FUNCTION_BLOCK MoveModuloMoverToPosition EXTENDS TaskBase
VAR_INPUT
END_VAR
VAR_OUTPUT
END_VAR
VAR
	moveAbs	: MC_MoveAbsoluteCA;
	_axis : REFERENCE TO AXIS_REF;
	_MoveMover : BOOL;
	_stOptions : ST_MoveAbsoluteCAOptions;
END_VAR

METHOD Abort : BOOL
moveAbs.Execute := FALSE;
moveAbs.Position := moveAbs.Velocity := 0;
_MoveMover := false;
_busy := false;
Abort := true;
State := 0;
END_METHOD

PROPERTY PUBLIC Acceleration : mc_lreal
GET
Acceleration := moveAbs.Acceleration;
END_GET
SET
moveAbs.Acceleration := Acceleration;
END_SET
END_PROPERTY

METHOD Cycle : BOOL
VAR_INPUT
END_VAR
CASE State OF
	0:
		IF _MoveMover THEN
			_done := FALSE;
			_error := FALSE;
			_busy := TRUE;
			moveAbs.Execute := TRUE;
			IF moveAbs.Busy THEN
				State := 10;
				_MoveMover := FALSE;
			END_IF
		END_IF
		
	10:
		IF NOT moveAbs.Busy THEN
			IF moveAbs.Done THEN
				_done := TRUE;
			ELSIF moveAbs.Error THEN
				_error := TRUE;
			END_IF
			_busy := FALSE;
			moveAbs.Execute := FALSE;
			State := 0;
		END_IF
END_CASE

moveAbs(Axis := _axis, Options := _stOptions);
END_METHOD

PROPERTY PUBLIC Deceleration : mc_lreal
GET
Deceleration := moveAbs.Deceleration;
END_GET
SET
moveAbs.Deceleration := Deceleration;
END_SET
END_PROPERTY

METHOD FB_init : BOOL
VAR_INPUT
	bInitRetains : BOOL; // if TRUE, the retain variables are initialized (warm start / cold start)
	bInCopyCode : BOOL;  // if TRUE, the instance afterwards gets moved into the copy code (online change)
	axis : reference TO AXIS_REF;
END_VAR
_axis REF= axis;
END_METHOD

PROPERTY PUBLIC Gap : mc_lreal
GET
Gap := moveAbs.Gap;
END_GET
SET
moveAbs.Gap := Gap;
END_SET
END_PROPERTY

PROPERTY PUBLIC Jerk : mc_lreal
GET
Jerk := moveAbs.Jerk;
END_GET
SET
moveAbs.Jerk := Jerk;
END_SET
END_PROPERTY

METHOD MoveTo : BOOL
VAR_INPUT
	Position : MC_LREAL;
	Velocity : MC_LREAL;
	Direction: Tc3_Mc3Definitions.MC_DIRECTION;
	Turns: UDINT;
END_VAR
moveAbs.Position := Position;
moveAbs.Velocity := Velocity;
moveAbs.Direction := Direction;
moveAbs.Options.AdditionalTurns := Turns;
_MoveMover := MoveTo := true;
END_METHOD

PROPERTY PUBLIC Options : ST_MoveAbsoluteCAOptions
GET
Options := _stOptions;
END_GET
SET
_stOptions := Options;
END_SET
END_PROPERTY

END_FUNCTION_BLOCK

(* stored: Version 1.1.0.1, ProductVersion 3.1.4024.12
   POU MoveModuloMoverToPosition: Id {996fe608-f005-43b0-b7bb-f33f237511c5}, SpecialFunc None
   Method Abort: Id {e91f53d6-3fee-47da-b969-b12290444a1f}
   Property Acceleration: Id {9cca71bc-09f7-4ec5-a9e0-372ce880866d}
   Get Get: Id {8efab319-7a15-4b02-96d3-afb30733e7b6}
   Set Set: Id {7f6e5164-788c-42d5-9777-9034d8aee40a}
   Method Cycle: Id {17422f94-11d5-4870-b9cb-2971dc153481}
   Property Deceleration: Id {844ebaf1-91dd-4442-8c33-92bcbeac6dea}
   Get Get: Id {50b8d5dc-c5e8-49f1-8033-680b16568e17}
   Set Set: Id {c1fd28c1-52e9-40a5-a51c-7d8bad271f43}
   Method FB_init: Id {37d409ee-dd67-4ea2-bddf-a65d46cc40e5}
   Property Gap: Id {1f9f5e65-07fb-4eac-aedb-feef80486e30}
   Get Get: Id {67ac09b0-11e2-4124-826d-72346d915abb}
   Set Set: Id {62c5bf39-3859-4737-8183-2c2206b5176d}
   Property Jerk: Id {cce85ebc-6201-45ef-a6f2-00296f696976}
   Get Get: Id {9dd7b014-e337-43e8-be50-6abb225db838}
   Set Set: Id {dcb14394-7c86-41b4-80fe-e9c7416faef5}
   Method MoveTo: Id {457265c4-5c25-4ff8-a5c9-719e58c0811a}
   Property Options: Id {c95271b4-8041-4fcf-9fb6-4915363c060f}
   Get Get: Id {965704cd-ef53-4074-a532-01335413067a}
   Set Set: Id {64fce6aa-8064-4054-b02a-ac33ceea4a73} *)
